//Extend the base errors with project errors
TYPE HMI_ERR_SafetyController1 EXTENDS HMI_ERR_SafetyLogic:
STRUCT
	//note: errors for inputs moved to input-instances
	;
END_STRUCT
END_TYPE

(* stored: Version 1.1.0.1
   DUT HMI_ERR_SafetyController1: Id {6e2c828e-75fe-07ca-202e-7bf6b613f847} *)
